{attribute addProperty BoxType "EL2596-0000-0017"}
{attribute addProperty Id "DOX_StatusAT %I*DOX_Status_95DEE7BC1620DOX_ControlAT %Q*DOX_Control_3320C5611620WcStateAT %I*WcState_98A4DF7520.250InfoDataAT %I*InfoData_BC63D37F80100"}
{attribute addProperty CRC "1250067191"}
{attribute addProperty SizeInBites "114"}
{attribute addProperty SizeInBytes "14.25"}
TYPE EL2596_81EB8F1B :
STRUCT
	{attribute addProperty Name "DOX_Status"}
	DOX_Status : DOX_Status_95DEE7BC;
	{attribute addProperty Name "DOX_Control"}
	DOX_Control : DOX_Control_3320C561;
	{attribute addProperty Name "WcState"}
	WcState : WcState_98A4DF75;
	{attribute addProperty Name "InfoData"}
	InfoData : InfoData_BC63D37F;
END_STRUCT
END_TYPE

(* stored: Version 1.2.0.0, ProductVersion 3.1.4024.9
   DUT EL2596_81EB8F1B: Id {52f59b52-e329-40ad-9ec6-ca92f66aa388} *)
